{attribute addProperty BoxType "EK1122-0000-0018"}
{attribute addProperty Id "Beckhoff_EP2xxxsub_EK1100EK1100_179A0949162A_0001_EP2001_1000_0016EP2001_62CCD7808811A_0002_EP2001_1000_0017EP2001_62CCD7808811A_0003_EP2001_1000_0018EP2001_62CCD7808811A_0004_EP2001_1000_0019EP2001_62CCD7808811A_0005_EP2008_0001_0016EP2008_04E0E56B8811A_0006_EP2008_0001_0017EP2008_04E0E56B8811A_0007_EP2008_0001_0018EP2008_04E0E56B8811A_0008_EP2008_0001_0019EP2008_04E0E56B8811A_0009_EP2008_0002_0016EP2008_04E0E56B8811A_0010_EP2008_0002_0017EP2008_04E0E56B8811A_0011_EP2008_0002_0018EP2008_04E0E56B8811A_0012_EP2008_0002_0019EP2008_04E0E56B8811A_0013_EP2008_0022_0016EP2008_04E0E56B8811A_0014_EP2008_0022_0017EP2008_04E0E56B8811A_0015_EP2008_0022_0018EP2008_04E0E56B8811A_0016_EP2028_0001_0016EP2028_04E0E56B8811A_0017_EP2028_0001_0017EP2028_04E0E56B8811A_0018_EP2028_0001_0018EP2028_04E0E56B8811A_0019_EP2028_0002_0016EP2028_04E0E56B8811A_0020_EP2028_0002_0017EP2028_04E0E56B8811A_0021_EP2028_0002_0018EP2028_04E0E56B8811A_0022_EP2028_0002_0019EP2028_04E0E56B8811A_0023_EP2028_0032_0017EP2028_04E0E56B8811A_0024_EP2028_0032_0018EP2028_04E0E56B8811A_0025_EP2028_0032_0019EP2028_04E0E56B8811A_0026_EP2038_0001_0016EP2038_309488D016020A_0027_EP2038_0001_0017EP2038_309488D016020A_0028_EP2038_0001_0018EP2038_309488D016020A_0029_EP2038_0002_0016EP2038_309488D016020A_0030_EP2038_0002_0017EP2038_309488D016020A_0031_EP2038_0002_0018EP2038_309488D016020A_0032_EP2308_0000_0016EP2308_E58483979612A_0033_EP2308_0000_0017EP2308_E58483979612A_0034_EP2308_0000_0018EP2308_E58483979612A_0035_EP2308_0001_0016EP2308_E58483979612A_0036_EP2308_0001_0017EP2308_E58483979612A_0037_EP2308_0001_0018EP2308_E58483979612A_0038_EP2308_0001_0019EP2308_E58483979612A_0039_EP2308_0002_0016EP2308_E58483979612A_0040_EP2308_0002_0017EP2308_E58483979612A_0041_EP2308_0002_0018EP2308_E58483979612A_0042_EP2308_0002_0019EP2308_E58483979612A_0043_EP2316_0003_0016EP2316_91349AC435244A_0044_EP2316_0003_0017EP2316_91349AC435244A_0045_EP2316_0003_0018EP2316_91349AC435244A_0046_EP2316_0008_0016EP2316_0F29F8B034443A_0047_EP2316_0008_0017EP2316_900F0E4A35244A_0048_EP2316_0008_0018EP2316_51C6E99B35244A_0049_EP2316_0008_0019EP2316_91349AC435244A_0050_EP2316_0008_0020EP2316_91349AC435244A_0051_EP2316_0008_0021EP2316_91349AC435244A_0052_EP2318_0001_0016EP2318_E58483979612A_0053_EP2318_0001_0017EP2318_E58483979612A_0054_EP2318_0001_0018EP2318_E58483979612A_0055_EP2318_0001_0019EP2318_E58483979612A_0056_EP2318_0002_0016EP2318_E58483979612A_0057_EP2318_0002_0017EP2318_E58483979612A_0058_EP2318_0002_0018EP2318_E58483979612A_0059_EP2318_0002_0019EP2318_E58483979612A_0060_EP2328_0001_0016EP2328_E58483979612A_0061_EP2328_0001_0017EP2328_E58483979612A_0062_EP2328_0001_0018EP2328_E58483979612A_0063_EP2328_0002_0016EP2328_E58483979612A_0064_EP2328_0002_0017EP2328_E58483979612A_0065_EP2328_0002_0018EP2328_E58483979612A_0066_EP2328_0002_0019EP2328_E58483979612A_0067_EP2328_1061_0016EP2328_6092ACCC9612A_0068_EP2338_0001_0016EP2338_584B274D16020A_0069_EP2338_0001_0017EP2338_584B274D16020A_0070_EP2338_0001_0018EP2338_6598BC3916020A_0071_EP2338_0001_0019EP2338_6598BC3916020A_0072_EP2338_0001_0020EP2338_6598BC3916020A_0073_EP2338_0001_0021EP2338_6598BC3916020A_0074_EP2338_0001_0022EP2338_6598BC3916020A_0075_EP2338_0001_0023EP2338_6598BC3916020A_0076_EP2338_0002_0016EP2338_584B274D16020A_0077_EP2338_0002_0017EP2338_584B274D16020A_0078_EP2338_0002_0018EP2338_6598BC3916020A_0079_EP2338_0002_0019EP2338_6598BC3916020A_0080_EP2338_0002_0020EP2338_6598BC3916020A_0081_EP2338_0002_0021EP2338_6598BC3916020A_0082_EP2338_0002_0022EP2338_6598BC3916020A_0083_EP2338_0002_0023EP2338_6598BC3916020A_0084_EP2338_1001_0016EP2338_6598BC3916020A_0085_EP2338_1001_0017EP2338_6598BC3916020A_0086_EP2338_1001_0018EP2338_6598BC3916020A_0087_EP2338_1002_0016EP2338_6598BC3916020A_0088_EP2338_1002_0017EP2338_6598BC3916020A_0089_EP2338_1002_0018EP2338_6598BC3916020A_0090_EP2339_0003_0016EP2339_CCF4B64340050A_0092_EP2339_0021_0016EP2339_C622991433642A_0093_EP2339_0021_0017EP2339_067D5D8B33642A_0094_EP2339_0021_0018EP2339_067D5D8B33642A_0095_EP2339_0021_0019EP2339_2F846F4A28836A_0096_EP2339_0021_0020EP2339_2F846F4A28836A_0097_EP2339_0022_0016EP2339_EFDBABD528836A_0098_EP2339_0022_0017EP2339_2F846F4A28836A_0099_EP2339_0022_0018EP2339_2F846F4A28836A_0100_EP2339_0022_0019EP2339_2F846F4A28836A_0101_EP2339_0042_0017EP2339_350240E09634359738380A_0102_EP2339_0042_0018EP2339_1E71110B429496720068719476724A_0103_EP2339_0121_0016EP2339_2F846F4A28836A_0104_EP2349_0021_0016EP2349_2F846F4A28836A_0105_EP2349_0021_0017EP2349_2F846F4A28836A_0106_EP2349_0021_0018EP2349_2F846F4A28836A_0107_EP2349_0022_0016EP2349_2F846F4A28836A_0108_EP2349_0022_0017EP2349_2F846F4A28836A_0109_EP2349_0022_0018EP2349_2F846F4A28836A_0110_EP2624_0002_0016EP2624_E7E37CC2567A_0111_EP2624_0002_0017EP2624_E7E37CC2567A_0112_EP2624_0002_0018EP2624_E7E37CC2567A_0113_EP2624_0002_0019EP2624_E7E37CC2567A_0114_EP2809_0021_0016EP2809_5A2A5F2915219A_0115_EP2809_0021_0017EP2809_5A2A5F2915219A_0116_EP2809_0021_0018EP2809_5A2A5F2915219A_0117_EP2809_0022_0016EP2809_5A2A5F2915219A_0118_EP2809_0022_0017EP2809_5A2A5F2915219A_0119_EP2809_0022_0018EP2809_5A2A5F2915219A_0120_EP2809_0042_0017EP2809_713014EC429496725634359738363A_0121_EP2809_0042_0018EP2809_F05176C6429496725634359738363A_0122_EP2816_0003_0016EP2816_D40507B840851A_0123_EP2816_0004_0016EP2816_0ADDCDDB21627A_0124_EP2816_0004_0017EP2816_D40507B840851A_0125_EP2816_0004_0018EP2816_D40507B840851A_0126_EP2816_0008_0016EP2816_B01EBB0F40851A_0127_EP2816_0008_0017EP2816_B01EBB0F40851A_0128_EP2816_0008_0018EP2816_C01896FF40851A_0129_EP2816_0008_0019EP2816_1A393DE740851A_0130_EP2816_0008_0020EP2816_1A393DE740851A_0131_EP2816_0008_0021EP2816_1A393DE740851A_0132_EP2816_0010_0016EP2816_B01EBB0F40851A_0133_EP2816_0010_0017EP2816_B01EBB0F40851A_0134_EP2816_0010_0018EP2816_C01896FF40851A_0135_EP2816_0010_0019EP2816_1A393DE740851A_0136_EP2816_0010_0020EP2816_1A393DE740851A_0137_EP2816_0010_0021EP2816_1A393DE740851A_0138_EP2817_0008_0016EP2817_A6BB1E3656070A_0139_EP2817_0008_0017EP2817_A6BB1E3656070A_0140_EP2817_0008_0018EP2817_A6BB1E3656070A_0141_EP2817_0008_0019EP2817_A6BB1E3656070"}
{attribute addProperty CRC "3275053809"}
{attribute addProperty SizeInBites "27232"}
{attribute addProperty SizeInBytes "171798695244"}
TYPE Beckhoff_EP2xxxEK1122_C3355AF1 EXTENDS EK1122_179A0949 :
STRUCT
	{attribute addProperty Name "Beckhoff_EP2xxxsub_EK1100"}
	Beckhoff_EP2xxxsub_EK1100 : EK1100_179A0949;
	{attribute addProperty Name "A_0001_EP2001_1000_0016"}
	A_0001_EP2001_1000_0016 : EP2001_62CCD780;
	{attribute addProperty Name "A_0002_EP2001_1000_0017"}
	A_0002_EP2001_1000_0017 : EP2001_62CCD780;
	{attribute addProperty Name "A_0003_EP2001_1000_0018"}
	A_0003_EP2001_1000_0018 : EP2001_62CCD780;
	{attribute addProperty Name "A_0004_EP2001_1000_0019"}
	A_0004_EP2001_1000_0019 : EP2001_62CCD780;
	{attribute addProperty Name "A_0005_EP2008_0001_0016"}
	A_0005_EP2008_0001_0016 : EP2008_04E0E56B;
	{attribute addProperty Name "A_0006_EP2008_0001_0017"}
	A_0006_EP2008_0001_0017 : EP2008_04E0E56B;
	{attribute addProperty Name "A_0007_EP2008_0001_0018"}
	A_0007_EP2008_0001_0018 : EP2008_04E0E56B;
	{attribute addProperty Name "A_0008_EP2008_0001_0019"}
	A_0008_EP2008_0001_0019 : EP2008_04E0E56B;
	{attribute addProperty Name "A_0009_EP2008_0002_0016"}
	A_0009_EP2008_0002_0016 : EP2008_04E0E56B;
	{attribute addProperty Name "A_0010_EP2008_0002_0017"}
	A_0010_EP2008_0002_0017 : EP2008_04E0E56B;
	{attribute addProperty Name "A_0011_EP2008_0002_0018"}
	A_0011_EP2008_0002_0018 : EP2008_04E0E56B;
	{attribute addProperty Name "A_0012_EP2008_0002_0019"}
	A_0012_EP2008_0002_0019 : EP2008_04E0E56B;
	{attribute addProperty Name "A_0013_EP2008_0022_0016"}
	A_0013_EP2008_0022_0016 : EP2008_04E0E56B;
	{attribute addProperty Name "A_0014_EP2008_0022_0017"}
	A_0014_EP2008_0022_0017 : EP2008_04E0E56B;
	{attribute addProperty Name "A_0015_EP2008_0022_0018"}
	A_0015_EP2008_0022_0018 : EP2008_04E0E56B;
	{attribute addProperty Name "A_0016_EP2028_0001_0016"}
	A_0016_EP2028_0001_0016 : EP2028_04E0E56B;
	{attribute addProperty Name "A_0017_EP2028_0001_0017"}
	A_0017_EP2028_0001_0017 : EP2028_04E0E56B;
	{attribute addProperty Name "A_0018_EP2028_0001_0018"}
	A_0018_EP2028_0001_0018 : EP2028_04E0E56B;
	{attribute addProperty Name "A_0019_EP2028_0002_0016"}
	A_0019_EP2028_0002_0016 : EP2028_04E0E56B;
	{attribute addProperty Name "A_0020_EP2028_0002_0017"}
	A_0020_EP2028_0002_0017 : EP2028_04E0E56B;
	{attribute addProperty Name "A_0021_EP2028_0002_0018"}
	A_0021_EP2028_0002_0018 : EP2028_04E0E56B;
	{attribute addProperty Name "A_0022_EP2028_0002_0019"}
	A_0022_EP2028_0002_0019 : EP2028_04E0E56B;
	{attribute addProperty Name "A_0023_EP2028_0032_0017"}
	A_0023_EP2028_0032_0017 : EP2028_04E0E56B;
	{attribute addProperty Name "A_0024_EP2028_0032_0018"}
	A_0024_EP2028_0032_0018 : EP2028_04E0E56B;
	{attribute addProperty Name "A_0025_EP2028_0032_0019"}
	A_0025_EP2028_0032_0019 : EP2028_04E0E56B;
	{attribute addProperty Name "A_0026_EP2038_0001_0016"}
	A_0026_EP2038_0001_0016 : EP2038_309488D0;
	{attribute addProperty Name "A_0027_EP2038_0001_0017"}
	A_0027_EP2038_0001_0017 : EP2038_309488D0;
	{attribute addProperty Name "A_0028_EP2038_0001_0018"}
	A_0028_EP2038_0001_0018 : EP2038_309488D0;
	{attribute addProperty Name "A_0029_EP2038_0002_0016"}
	A_0029_EP2038_0002_0016 : EP2038_309488D0;
	{attribute addProperty Name "A_0030_EP2038_0002_0017"}
	A_0030_EP2038_0002_0017 : EP2038_309488D0;
	{attribute addProperty Name "A_0031_EP2038_0002_0018"}
	A_0031_EP2038_0002_0018 : EP2038_309488D0;
	{attribute addProperty Name "A_0032_EP2308_0000_0016"}
	A_0032_EP2308_0000_0016 : EP2308_E5848397;
	{attribute addProperty Name "A_0033_EP2308_0000_0017"}
	A_0033_EP2308_0000_0017 : EP2308_E5848397;
	{attribute addProperty Name "A_0034_EP2308_0000_0018"}
	A_0034_EP2308_0000_0018 : EP2308_E5848397;
	{attribute addProperty Name "A_0035_EP2308_0001_0016"}
	A_0035_EP2308_0001_0016 : EP2308_E5848397;
	{attribute addProperty Name "A_0036_EP2308_0001_0017"}
	A_0036_EP2308_0001_0017 : EP2308_E5848397;
	{attribute addProperty Name "A_0037_EP2308_0001_0018"}
	A_0037_EP2308_0001_0018 : EP2308_E5848397;
	{attribute addProperty Name "A_0038_EP2308_0001_0019"}
	A_0038_EP2308_0001_0019 : EP2308_E5848397;
	{attribute addProperty Name "A_0039_EP2308_0002_0016"}
	A_0039_EP2308_0002_0016 : EP2308_E5848397;
	{attribute addProperty Name "A_0040_EP2308_0002_0017"}
	A_0040_EP2308_0002_0017 : EP2308_E5848397;
	{attribute addProperty Name "A_0041_EP2308_0002_0018"}
	A_0041_EP2308_0002_0018 : EP2308_E5848397;
	{attribute addProperty Name "A_0042_EP2308_0002_0019"}
	A_0042_EP2308_0002_0019 : EP2308_E5848397;
	{attribute addProperty Name "A_0043_EP2316_0003_0016"}
	A_0043_EP2316_0003_0016 : EP2316_91349AC4;
	{attribute addProperty Name "A_0044_EP2316_0003_0017"}
	A_0044_EP2316_0003_0017 : EP2316_91349AC4;
	{attribute addProperty Name "A_0045_EP2316_0003_0018"}
	A_0045_EP2316_0003_0018 : EP2316_91349AC4;
	{attribute addProperty Name "A_0046_EP2316_0008_0016"}
	A_0046_EP2316_0008_0016 : EP2316_0F29F8B0;
	{attribute addProperty Name "A_0047_EP2316_0008_0017"}
	A_0047_EP2316_0008_0017 : EP2316_900F0E4A;
	{attribute addProperty Name "A_0048_EP2316_0008_0018"}
	A_0048_EP2316_0008_0018 : EP2316_51C6E99B;
	{attribute addProperty Name "A_0049_EP2316_0008_0019"}
	A_0049_EP2316_0008_0019 : EP2316_91349AC4;
	{attribute addProperty Name "A_0050_EP2316_0008_0020"}
	A_0050_EP2316_0008_0020 : EP2316_91349AC4;
	{attribute addProperty Name "A_0051_EP2316_0008_0021"}
	A_0051_EP2316_0008_0021 : EP2316_91349AC4;
	{attribute addProperty Name "A_0052_EP2318_0001_0016"}
	A_0052_EP2318_0001_0016 : EP2318_E5848397;
	{attribute addProperty Name "A_0053_EP2318_0001_0017"}
	A_0053_EP2318_0001_0017 : EP2318_E5848397;
	{attribute addProperty Name "A_0054_EP2318_0001_0018"}
	A_0054_EP2318_0001_0018 : EP2318_E5848397;
	{attribute addProperty Name "A_0055_EP2318_0001_0019"}
	A_0055_EP2318_0001_0019 : EP2318_E5848397;
	{attribute addProperty Name "A_0056_EP2318_0002_0016"}
	A_0056_EP2318_0002_0016 : EP2318_E5848397;
	{attribute addProperty Name "A_0057_EP2318_0002_0017"}
	A_0057_EP2318_0002_0017 : EP2318_E5848397;
	{attribute addProperty Name "A_0058_EP2318_0002_0018"}
	A_0058_EP2318_0002_0018 : EP2318_E5848397;
	{attribute addProperty Name "A_0059_EP2318_0002_0019"}
	A_0059_EP2318_0002_0019 : EP2318_E5848397;
	{attribute addProperty Name "A_0060_EP2328_0001_0016"}
	A_0060_EP2328_0001_0016 : EP2328_E5848397;
	{attribute addProperty Name "A_0061_EP2328_0001_0017"}
	A_0061_EP2328_0001_0017 : EP2328_E5848397;
	{attribute addProperty Name "A_0062_EP2328_0001_0018"}
	A_0062_EP2328_0001_0018 : EP2328_E5848397;
	{attribute addProperty Name "A_0063_EP2328_0002_0016"}
	A_0063_EP2328_0002_0016 : EP2328_E5848397;
	{attribute addProperty Name "A_0064_EP2328_0002_0017"}
	A_0064_EP2328_0002_0017 : EP2328_E5848397;
	{attribute addProperty Name "A_0065_EP2328_0002_0018"}
	A_0065_EP2328_0002_0018 : EP2328_E5848397;
	{attribute addProperty Name "A_0066_EP2328_0002_0019"}
	A_0066_EP2328_0002_0019 : EP2328_E5848397;
	{attribute addProperty Name "A_0067_EP2328_1061_0016"}
	A_0067_EP2328_1061_0016 : EP2328_6092ACCC;
	{attribute addProperty Name "A_0068_EP2338_0001_0016"}
	A_0068_EP2338_0001_0016 : EP2338_584B274D;
	{attribute addProperty Name "A_0069_EP2338_0001_0017"}
	A_0069_EP2338_0001_0017 : EP2338_584B274D;
	{attribute addProperty Name "A_0070_EP2338_0001_0018"}
	A_0070_EP2338_0001_0018 : EP2338_6598BC39;
	{attribute addProperty Name "A_0071_EP2338_0001_0019"}
	A_0071_EP2338_0001_0019 : EP2338_6598BC39;
	{attribute addProperty Name "A_0072_EP2338_0001_0020"}
	A_0072_EP2338_0001_0020 : EP2338_6598BC39;
	{attribute addProperty Name "A_0073_EP2338_0001_0021"}
	A_0073_EP2338_0001_0021 : EP2338_6598BC39;
	{attribute addProperty Name "A_0074_EP2338_0001_0022"}
	A_0074_EP2338_0001_0022 : EP2338_6598BC39;
	{attribute addProperty Name "A_0075_EP2338_0001_0023"}
	A_0075_EP2338_0001_0023 : EP2338_6598BC39;
	{attribute addProperty Name "A_0076_EP2338_0002_0016"}
	A_0076_EP2338_0002_0016 : EP2338_584B274D;
	{attribute addProperty Name "A_0077_EP2338_0002_0017"}
	A_0077_EP2338_0002_0017 : EP2338_584B274D;
	{attribute addProperty Name "A_0078_EP2338_0002_0018"}
	A_0078_EP2338_0002_0018 : EP2338_6598BC39;
	{attribute addProperty Name "A_0079_EP2338_0002_0019"}
	A_0079_EP2338_0002_0019 : EP2338_6598BC39;
	{attribute addProperty Name "A_0080_EP2338_0002_0020"}
	A_0080_EP2338_0002_0020 : EP2338_6598BC39;
	{attribute addProperty Name "A_0081_EP2338_0002_0021"}
	A_0081_EP2338_0002_0021 : EP2338_6598BC39;
	{attribute addProperty Name "A_0082_EP2338_0002_0022"}
	A_0082_EP2338_0002_0022 : EP2338_6598BC39;
	{attribute addProperty Name "A_0083_EP2338_0002_0023"}
	A_0083_EP2338_0002_0023 : EP2338_6598BC39;
	{attribute addProperty Name "A_0084_EP2338_1001_0016"}
	A_0084_EP2338_1001_0016 : EP2338_6598BC39;
	{attribute addProperty Name "A_0085_EP2338_1001_0017"}
	A_0085_EP2338_1001_0017 : EP2338_6598BC39;
	{attribute addProperty Name "A_0086_EP2338_1001_0018"}
	A_0086_EP2338_1001_0018 : EP2338_6598BC39;
	{attribute addProperty Name "A_0087_EP2338_1002_0016"}
	A_0087_EP2338_1002_0016 : EP2338_6598BC39;
	{attribute addProperty Name "A_0088_EP2338_1002_0017"}
	A_0088_EP2338_1002_0017 : EP2338_6598BC39;
	{attribute addProperty Name "A_0089_EP2338_1002_0018"}
	A_0089_EP2338_1002_0018 : EP2338_6598BC39;
	{attribute addProperty Name "A_0090_EP2339_0003_0016"}
	A_0090_EP2339_0003_0016 : EP2339_CCF4B643;
	{attribute addProperty Name "A_0092_EP2339_0021_0016"}
	A_0092_EP2339_0021_0016 : EP2339_C6229914;
	{attribute addProperty Name "A_0093_EP2339_0021_0017"}
	A_0093_EP2339_0021_0017 : EP2339_067D5D8B;
	{attribute addProperty Name "A_0094_EP2339_0021_0018"}
	A_0094_EP2339_0021_0018 : EP2339_067D5D8B;
	{attribute addProperty Name "A_0095_EP2339_0021_0019"}
	A_0095_EP2339_0021_0019 : EP2339_2F846F4A;
	{attribute addProperty Name "A_0096_EP2339_0021_0020"}
	A_0096_EP2339_0021_0020 : EP2339_2F846F4A;
	{attribute addProperty Name "A_0097_EP2339_0022_0016"}
	A_0097_EP2339_0022_0016 : EP2339_EFDBABD5;
	{attribute addProperty Name "A_0098_EP2339_0022_0017"}
	A_0098_EP2339_0022_0017 : EP2339_2F846F4A;
	{attribute addProperty Name "A_0099_EP2339_0022_0018"}
	A_0099_EP2339_0022_0018 : EP2339_2F846F4A;
	{attribute addProperty Name "A_0100_EP2339_0022_0019"}
	A_0100_EP2339_0022_0019 : EP2339_2F846F4A;
	{attribute addProperty Name "A_0101_EP2339_0042_0017"}
	A_0101_EP2339_0042_0017 : EP2339_350240E0;
	{attribute addProperty Name "A_0102_EP2339_0042_0018"}
	A_0102_EP2339_0042_0018 : EP2339_1E71110B;
	{attribute addProperty Name "A_0103_EP2339_0121_0016"}
	A_0103_EP2339_0121_0016 : EP2339_2F846F4A;
	{attribute addProperty Name "A_0104_EP2349_0021_0016"}
	A_0104_EP2349_0021_0016 : EP2349_2F846F4A;
	{attribute addProperty Name "A_0105_EP2349_0021_0017"}
	A_0105_EP2349_0021_0017 : EP2349_2F846F4A;
	{attribute addProperty Name "A_0106_EP2349_0021_0018"}
	A_0106_EP2349_0021_0018 : EP2349_2F846F4A;
	{attribute addProperty Name "A_0107_EP2349_0022_0016"}
	A_0107_EP2349_0022_0016 : EP2349_2F846F4A;
	{attribute addProperty Name "A_0108_EP2349_0022_0017"}
	A_0108_EP2349_0022_0017 : EP2349_2F846F4A;
	{attribute addProperty Name "A_0109_EP2349_0022_0018"}
	A_0109_EP2349_0022_0018 : EP2349_2F846F4A;
	{attribute addProperty Name "A_0110_EP2624_0002_0016"}
	A_0110_EP2624_0002_0016 : EP2624_E7E37CC2;
	{attribute addProperty Name "A_0111_EP2624_0002_0017"}
	A_0111_EP2624_0002_0017 : EP2624_E7E37CC2;
	{attribute addProperty Name "A_0112_EP2624_0002_0018"}
	A_0112_EP2624_0002_0018 : EP2624_E7E37CC2;
	{attribute addProperty Name "A_0113_EP2624_0002_0019"}
	A_0113_EP2624_0002_0019 : EP2624_E7E37CC2;
	{attribute addProperty Name "A_0114_EP2809_0021_0016"}
	A_0114_EP2809_0021_0016 : EP2809_5A2A5F29;
	{attribute addProperty Name "A_0115_EP2809_0021_0017"}
	A_0115_EP2809_0021_0017 : EP2809_5A2A5F29;
	{attribute addProperty Name "A_0116_EP2809_0021_0018"}
	A_0116_EP2809_0021_0018 : EP2809_5A2A5F29;
	{attribute addProperty Name "A_0117_EP2809_0022_0016"}
	A_0117_EP2809_0022_0016 : EP2809_5A2A5F29;
	{attribute addProperty Name "A_0118_EP2809_0022_0017"}
	A_0118_EP2809_0022_0017 : EP2809_5A2A5F29;
	{attribute addProperty Name "A_0119_EP2809_0022_0018"}
	A_0119_EP2809_0022_0018 : EP2809_5A2A5F29;
	{attribute addProperty Name "A_0120_EP2809_0042_0017"}
	A_0120_EP2809_0042_0017 : EP2809_713014EC;
	{attribute addProperty Name "A_0121_EP2809_0042_0018"}
	A_0121_EP2809_0042_0018 : EP2809_F05176C6;
	{attribute addProperty Name "A_0122_EP2816_0003_0016"}
	A_0122_EP2816_0003_0016 : EP2816_D40507B8;
	{attribute addProperty Name "A_0123_EP2816_0004_0016"}
	A_0123_EP2816_0004_0016 : EP2816_0ADDCDDB;
	{attribute addProperty Name "A_0124_EP2816_0004_0017"}
	A_0124_EP2816_0004_0017 : EP2816_D40507B8;
	{attribute addProperty Name "A_0125_EP2816_0004_0018"}
	A_0125_EP2816_0004_0018 : EP2816_D40507B8;
	{attribute addProperty Name "A_0126_EP2816_0008_0016"}
	A_0126_EP2816_0008_0016 : EP2816_B01EBB0F;
	{attribute addProperty Name "A_0127_EP2816_0008_0017"}
	A_0127_EP2816_0008_0017 : EP2816_B01EBB0F;
	{attribute addProperty Name "A_0128_EP2816_0008_0018"}
	A_0128_EP2816_0008_0018 : EP2816_C01896FF;
	{attribute addProperty Name "A_0129_EP2816_0008_0019"}
	A_0129_EP2816_0008_0019 : EP2816_1A393DE7;
	{attribute addProperty Name "A_0130_EP2816_0008_0020"}
	A_0130_EP2816_0008_0020 : EP2816_1A393DE7;
	{attribute addProperty Name "A_0131_EP2816_0008_0021"}
	A_0131_EP2816_0008_0021 : EP2816_1A393DE7;
	{attribute addProperty Name "A_0132_EP2816_0010_0016"}
	A_0132_EP2816_0010_0016 : EP2816_B01EBB0F;
	{attribute addProperty Name "A_0133_EP2816_0010_0017"}
	A_0133_EP2816_0010_0017 : EP2816_B01EBB0F;
	{attribute addProperty Name "A_0134_EP2816_0010_0018"}
	A_0134_EP2816_0010_0018 : EP2816_C01896FF;
	{attribute addProperty Name "A_0135_EP2816_0010_0019"}
	A_0135_EP2816_0010_0019 : EP2816_1A393DE7;
	{attribute addProperty Name "A_0136_EP2816_0010_0020"}
	A_0136_EP2816_0010_0020 : EP2816_1A393DE7;
	{attribute addProperty Name "A_0137_EP2816_0010_0021"}
	A_0137_EP2816_0010_0021 : EP2816_1A393DE7;
	{attribute addProperty Name "A_0138_EP2817_0008_0016"}
	A_0138_EP2817_0008_0016 : EP2817_A6BB1E36;
	{attribute addProperty Name "A_0139_EP2817_0008_0017"}
	A_0139_EP2817_0008_0017 : EP2817_A6BB1E36;
	{attribute addProperty Name "A_0140_EP2817_0008_0018"}
	A_0140_EP2817_0008_0018 : EP2817_A6BB1E36;
	{attribute addProperty Name "A_0141_EP2817_0008_0019"}
	A_0141_EP2817_0008_0019 : EP2817_A6BB1E36;
END_STRUCT
END_TYPE

(* stored: Version 1.2.0.0, ProductVersion 3.1.4024.9
   DUT Beckhoff_EP2xxxEK1122_C3355AF1: Id {b6781988-0df8-48c6-b6cc-ff0e7cb75515} *)
